FUNCTION_BLOCK Area_CAT_HMI (* Service Interface Function Block Type *)
  (* Standard: 61499-2 *)
  (* Version 0.0, 7/23/2025, Evans_A, Schneider Electric, template *)
  PACKAGE Main;
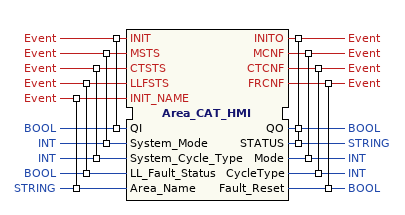
  EVENT_INPUT
    INIT WITH QI;
    MSTS WITH System_Mode;
    CTSTS WITH System_Cycle_Type;
    LLFSTS WITH LL_Fault_Status;
    INIT_NAME WITH Area_Name;
  END_EVENT
  EVENT_OUTPUT
    INITO WITH QO, STATUS;
    MCNF WITH Mode;
    CTCNF WITH CycleType;
    FRCNF WITH Fault_Reset;
  END_EVENT
  VAR_INPUT
    QI : BOOL;
    System_Mode : INT;
    System_Cycle_Type : INT;
    LL_Fault_Status : BOOL;
    Area_Name : STRING;
  END_VAR
  VAR_OUTPUT
    QO : BOOL; (* Event Output Qualifier *)
    STATUS : STRING; (* Service Status *)
    Mode : INT;
    CycleType : INT;
    Fault_Reset : BOOL;
  END_VAR
  SERVICE /
    SEQUENCE 
    END_SEQUENCE
  END_SERVICE
END_FUNCTION_BLOCK
